PROGRAM Axis01_Interlock_ST
VAR
    Always_ON  : BOOL := TRUE;
    Always_OFF : BOOL := FALSE;
END_VAR

IF (GVL_Axis02.Real_Position <= 55.0) THEN
	GVL_Axis01.Interlock := TRUE;
ELSIF GVL_Axis01.Command_Data > 0.0 THEN
		GVL_Axis01.Interlock := True;
END_IF

END_PROGRAM

(* stored: Version 1.1.0.1, ProductVersion 3.1.4024.15
   POU Axis01_Interlock_ST: Id {96374503-6a3b-4b57-9ef7-1c04f04096f0}, SpecialFunc None *)
